# EPICS autosave request: 3-0/GalilSup/Db/galil_ctrl_extras.req
# Controller settings
$(P)LIMITTYPE_CMD.VAL
$(P)HOMETYPE_CMD.VAL
